{attribute 'qualified_only'}
VAR_GLOBAL
	senNO				: FB_Sensor_NO;
	senNC				: FB_Sensor_NC;
	senNO_2inRow		: FB_Sensor_NO_2InRow;
	
	senNO_TestDecorator			: FB_Sensor_NO_TestDecorator (fbToDecorate := senNO);
	senNC_TestDecorator			: FB_Sensor_NC_TestDecorator (fbToDecorate := senNC);
	senNO_2inRow_TestDecorator	: FB_Sensor_NO_2InRow_TestDecorator (fbToDecorate := senNO_2inRow);
	
	
	senActuator1Start		: FB_Sensor_NO;
	senActuator1End			: FB_Sensor_NO;
	evActuator1				: FB_Electrovalve_5on2_1Coil;

	senActuator1Start_TestCecorator		: FB_Sensor_NO_TestDecorator (fbToDecorate := senActuator1Start);
	senActuator1End_TestDecorator		: FB_Sensor_NO_TestDecorator (fbToDecorate := senActuator1End);
	
	actActuator1			: FB_Actuator (
								senStart	:= senActuator1Start_TestCecorator,
								senEnd		:= senActuator1End_TestDecorator,
								evControl	:= evActuator1
							);
	
	actActuator1_TestWithoutTimeDecorator	: FB_Actuator_TestWithoutTimeDecorator (
											fbToDecorate	:= actActuator1,
											actActuator		:= actActuator1,
											senStart		:= senActuator1Start_TestCecorator,
											senEnd			:= senActuator1End_TestDecorator
										);
	

	actActuator1_TestWithTimeDecorator	: FB_Actuator_TestWithTimeDecorator (
											fbToDecorate	:= actActuator1,
											actActuator		:= actActuator1,
											senStart		:= senActuator1Start_TestCecorator,
											senEnd			:= senActuator1End_TestDecorator
										);
	flSS1						: FB_BaseFlag;
	flSTO						: FB_BaseFlag;
	fbLogger					: FB_BaseLogger;
	fbTime						: FB_BaseTime;
	fbLocaciotn					: FB_BaseLocation;	
	stCommonData				: ST_BaseCommonData;
	
END_VAR

(* stored: Version 1.1.0.1
   GVL GVL_Decorators: Id {93801117-c7f4-0fb3-1aa6-e6d5619250c7} *)
